INTERFACE I_HE_SolidAttenuatorHolder EXTENDS I_Fallible

METHOD GetMaterialAtBeamPosition
VAR_INPUT
END_VAR
END_METHOD

METHOD GetThicknessAtBeamPosition
VAR_INPUT
END_VAR
END_METHOD


METHOD HasSpecifiedFilter : BOOL
VAR_INPUT
    Filter : I_HE_SolidAttenuatorFilter;
END_VAR
END_METHOD


METHOD MoveToSpecifiedSlot
VAR_INPUT
    Slot : I_HE_SolidAttenuatorSlot;
    OffsetFromCenter : I_QuantityLREAL;
END_VAR
END_METHOD

END_INTERFACE

(* stored: Version 1.1.0.1
   Itf I_HE_SolidAttenuatorHolder: Id {8770de0e-d2e8-43c9-99d9-0c582407d0e4}
   Method GetMaterialAtBeamPosition: Id {4a113ab0-ee86-49ac-adfa-371a12e72394}
   Method GetThicknessAtBeamPosition: Id {3ad15a3b-3cef-43ef-b7ea-bbf762190556}
   Method HasSpecifiedFilter: Id {a23d5435-1469-4ae4-ab2f-fc9ea447fce6}
   Method MoveToSpecifiedSlot: Id {22088386-2d16-45d1-a254-d8397f1ac80e} *)
